FUNCTION_BLOCK FB_NOTT_CRYO_CTRL
VAR_INPUT
END_VAR
VAR_OUTPUT
END_VAR
VAR
	
	temp_1:		FB_CRYO_SENSOR_TEMPERATURE;
	temp_2:		FB_CRYO_SENSOR_TEMPERATURE;
	temp_3:		FB_CRYO_SENSOR_TEMPERATURE;
	temp_4:		FB_CRYO_SENSOR_TEMPERATURE;
	{attribute 'OPC.UA.DA' := '1'}
	lrTempC_1:	LREAL;
	{attribute 'OPC.UA.DA' := '1'}
	lrTempC_2:	LREAL;
	{attribute 'OPC.UA.DA' := '1'}
	lrTempC_3:	LREAL;
	{attribute 'OPC.UA.DA' := '1'}
	lrTempC_4:	LREAL;
END_VAR


M_ReadSensors();

METHOD M_ReadSensors
VAR_INPUT
END_VAR
temp_1(
	in_sName:= 'Temp 1', 
	in_nType:= E_CRYO_SENSOR_TYPE_TEMP.PT100, 
	in_lrScale:= 0.1, 
	in_bIgnoreUnderrange:= TRUE, 
	in_nRampPeriodSec:= 60, 
	in_bResistor_1_64:= );
lrTempC_1 := temp_1.stat.lrTempC;	

temp_2(
	in_sName:= 'Temp 2', 
	in_nType:= E_CRYO_SENSOR_TYPE_TEMP.PT100, 
	in_lrScale:= 0.1, 
	in_bIgnoreUnderrange:= TRUE, 
	in_nRampPeriodSec:= 60, 
	in_bResistor_1_64:= );
lrTempC_2 := temp_2.stat.lrTempC;
	
temp_3(
	in_sName:= 'Temp 3', 
	in_nType:= E_CRYO_SENSOR_TYPE_TEMP.PT100, 
	in_lrScale:= 0.1, 
	in_bIgnoreUnderrange:= TRUE, 
	in_nRampPeriodSec:= 60, 
	in_bResistor_1_64:= );
lrTempC_3 := temp_3.stat.lrTempC;
	
temp_4(
	in_sName:= 'Temp 4', 
	in_nType:= E_CRYO_SENSOR_TYPE_TEMP.PT100, 
	in_lrScale:= 0.1, 
	in_bIgnoreUnderrange:= TRUE, 
	in_nRampPeriodSec:= 60, 
	in_bResistor_1_64:= );
lrTempC_4 := temp_4.stat.lrTempC;
END_METHOD

END_FUNCTION_BLOCK

(* stored: Version 1.1.0.1, ProductVersion 3.1.4024.15
   POU FB_NOTT_CRYO_CTRL: Id {6db86964-7275-49aa-8bde-6c64e8e92208}, SpecialFunc None
   Method M_ReadSensors: Id {55b09f23-1072-4390-9e1d-acc3ae7e70c2} *)
